// TIA Portal project "AutoCrib_StMartin" (V19)

(* hardware
DEVICE "S7-1200 station_1"  S7-1200 Station
   slot 0: "Rack_0"  S7-1200 Rack  Rack  V1.0
   slot 1: "AutoCrib_PLC"  CPU 1215C AC/DC/Rly  6ES7 215-1BG40-0XB0  V4.6
*)

// ===== PLC "AutoCrib_PLC"  CPU 1215C AC/DC/Rly =====

VAR_GLOBAL   // PLC tag table "Tt_AdminPanel"
   "xAutomaticMode" AT %I0.5 : Bool;
   "xModeChangeButton" AT %I0.4 : Bool;
END_VAR

VAR_GLOBAL   // PLC tag table "Tt_UserPanel"
   "IX_CoinSensor" AT %I0.1 : Bool;
   "IX_Billsensor" AT %I0.3 : Bool;
   "IX_MotionSensor" AT %I0.0 : Bool;
   "IX_CoinSensorCrib" AT %I0.2 : Bool;
END_VAR

VAR_GLOBAL   // PLC tag table "Tt_LightGroups"
   "QX_MinimalLightGroup" AT %Q0.0 : Bool;
   "QX_MinimalPlusLightGroup" AT %Q0.1 : Bool;
   "QX_LightGroup1" AT %Q0.2 : Bool;
   "QX_LightGroup2" AT %Q0.3 : Bool;
   "QX_LightGroup3" AT %Q0.4 : Bool;
   "QX_LightGroup4" AT %Q0.5 : Bool;
   "QX_LightGroup5" AT %Q0.6 : Bool;
   "QX_LightGroup6" AT %Q0.7 : Bool;
   "QX_LightGroup7" AT %Q1.0 : Bool;
   "QX_LightGroup_Fire" AT %Q1.1 : Bool;
END_VAR

TYPE "DT_TimeConfig"
   STRUCT
      TOD_WakeUpTime : Time_Of_Day := TOD#08:00:00;
      TOD_SleepTime : Time_Of_Day := TOD#20:00:00;
   END_STRUCT;
END_TYPE

DATA_BLOCK "DB_Global_Time"   // DB2
{ S7_Optimized_Access := 'TRUE' }
VERSION : 0.1
   VAR
      DTL_CurrentTime : DTL;
      currentDate : Date;
      TOD_CurrentTime : Time_Of_Day;
      iDayTimeError : Int;
      xDayTime : Bool := False;
      tCycleTimePT : Time := T#20S;
      tShortCycleTimePT : Time := T#2S;
      tNoMotionTimeOut : Time := T#100S;
      tSystemEnable : "DT_TimeConfig";
   END_VAR
BEGIN
   tSystemEnable.TOD_WakeUpTime := TOD#08:00:00;
   tSystemEnable.TOD_SleepTime := TOD#19:00:00;
END_DATA_BLOCK

DATA_BLOCK "DB_Global_Config"   // DB8
{ S7_Optimized_Access := 'TRUE' }
VERSION : 0.1
BEGIN
END_DATA_BLOCK

// folder: FunctionBlocks

DATA_BLOCK "FB_Time_Update_DB"   // DB1
{ S7_Optimized_Access := 'TRUE' }
VERSION : 0.1
// stored: InstanceOfName FB_Time_Update
"FB_Time_Update"
BEGIN
END_DATA_BLOCK

// folder: FunctionBlocks/MainStateMachine

DATA_BLOCK "FB_MainStateMachine_DB"   // DB7
{ S7_Optimized_Access := 'TRUE' }
VERSION : 0.1
// stored: InstanceOfName FB_MainStateMachine
"FB_MainStateMachine"
BEGIN
END_DATA_BLOCK

// folder: System blocks/Program resources

DATA_BLOCK "IEC_Timer_0_DB_AutoChangeLighting"   // DB6
{ S7_Optimized_Access := 'TRUE' }
AUTHOR : Simatic
FAMILY : IEC
NAME : IEC_TMR
VERSION : 1.0
// stored: InstanceOfName IEC_TIMER
"IEC_TIMER"
BEGIN
END_DATA_BLOCK

// folder: (top level)

FUNCTION "checkForChristmas" : Bool   // FC1, SCL
{ S7_Optimized_Access := 'TRUE' }
VERSION : 0.1
   VAR_INPUT
      inputDate : Date;
   END_VAR
   VAR_TEMP
      iCurrentDate : Int;
      iCurrentMonth : Int;
      iCurrentDay : Int;
   END_VAR
BEGIN
   #iCurrentDate := DATE_TO_INT(#inputDate);

   // Extract month and day
   #iCurrentMonth := (#iCurrentDate / 100) MOD 100;  // Get the month (MM)
   #iCurrentDay := #iCurrentDate MOD 100;  // Get the day (DD)

   // Check if the date is December 24th
   IF (#iCurrentMonth = 12) AND (#iCurrentDay = 24) THEN
       // Date is December 24th
       #checkForChristmas := TRUE;
   END_IF;
END_FUNCTION

ORGANIZATION_BLOCK "Main"   // OB1, LAD, ProgramCycle
TITLE = "Main Program Sweep (Cycle)"
{ S7_Optimized_Access := 'TRUE' }
VERSION : 0.1
// Copyright to - B.Eng Ben Cloos - ben(at)cloosefamill.lu
   VAR_INPUT
      Initial_Call : Bool;   // Initial call of this OB
      Remanence : Bool;   // =True, if remanent data are available
   END_VAR
   VAR_TEMP
      xRT_CoinSensorTriggerQ : Bool;
      xRT_BillSensorTriggerQ : Bool;
      xRT_ModeChangeTriggerQ : Bool;
      xRT_MotionTriggerQ : Bool;
      b_IsChristmas : Bool;
   END_VAR
BEGIN

REGION Network 1: Update Time every Cycle
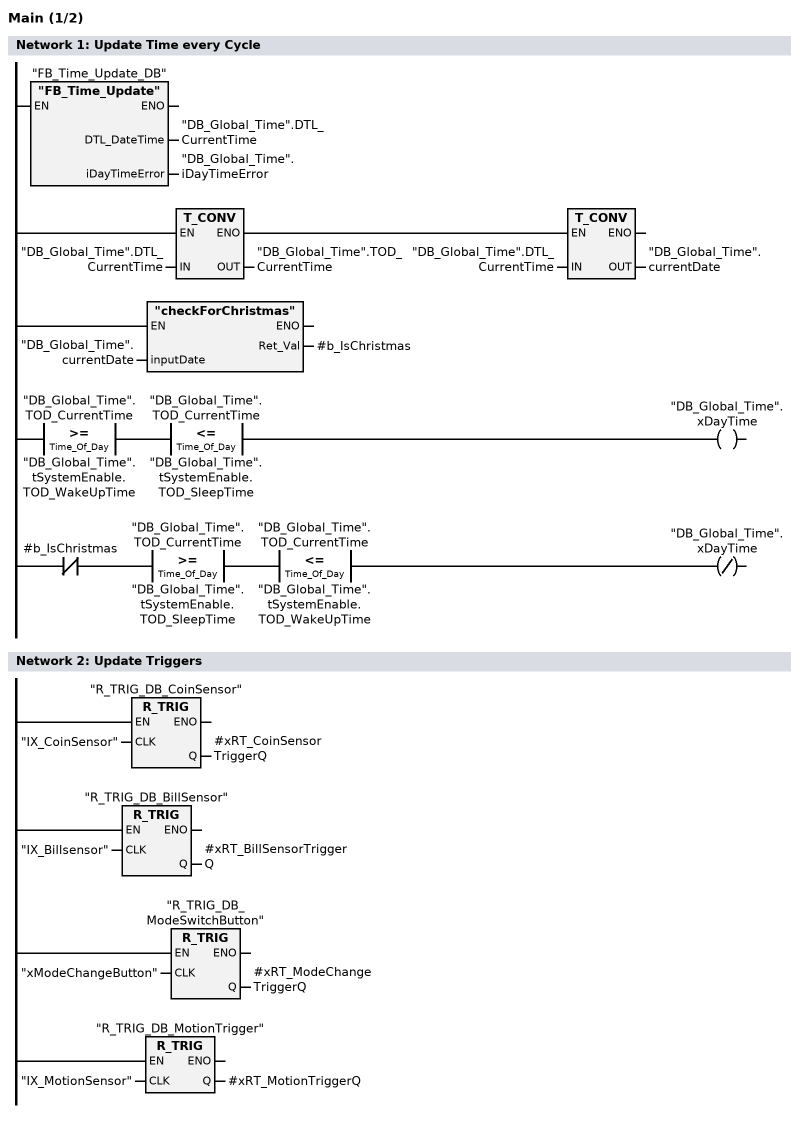
   // ENO of a box is taken as its EN; it also drops when the box reports an error
   "FB_Time_Update_DB"(DTL_DateTime => "DB_Global_Time".DTL_CurrentTime,   // "FB_Time_Update"
                       iDayTimeError => "DB_Global_Time".iDayTimeError);
   "DB_Global_Time".TOD_CurrentTime := T_CONV(IN := "DB_Global_Time".DTL_CurrentTime);
   "DB_Global_Time".currentDate := T_CONV(IN := "DB_Global_Time".DTL_CurrentTime);
   #b_IsChristmas := "checkForChristmas"(inputDate := "DB_Global_Time".currentDate);
   "DB_Global_Time".xDayTime := ("DB_Global_Time".TOD_CurrentTime >= "DB_Global_Time".tSystemEnable.TOD_WakeUpTime) AND ("DB_Global_Time".TOD_CurrentTime <= "DB_Global_Time".tSystemEnable.TOD_SleepTime);
   "DB_Global_Time".xDayTime := NOT (NOT #b_IsChristmas AND ("DB_Global_Time".TOD_CurrentTime >= "DB_Global_Time".tSystemEnable.TOD_SleepTime) AND ("DB_Global_Time".TOD_CurrentTime <= "DB_Global_Time".tSystemEnable.TOD_WakeUpTime));
END_REGION

REGION Network 2: Update Triggers
   "R_TRIG_DB_CoinSensor"(CLK := "IX_CoinSensor", Q => #xRT_CoinSensorTriggerQ);   // R_TRIG
   "R_TRIG_DB_BillSensor"(CLK := "IX_Billsensor", Q => #xRT_BillSensorTriggerQ);   // R_TRIG
   "R_TRIG_DB_ModeSwitchButton"(CLK := "xModeChangeButton", Q => #xRT_ModeChangeTriggerQ);   // R_TRIG
   "R_TRIG_DB_MotionTrigger"(CLK := "IX_MotionSensor", Q => #xRT_MotionTriggerQ);   // R_TRIG
END_REGION

REGION Network 3: State Machine Excecution
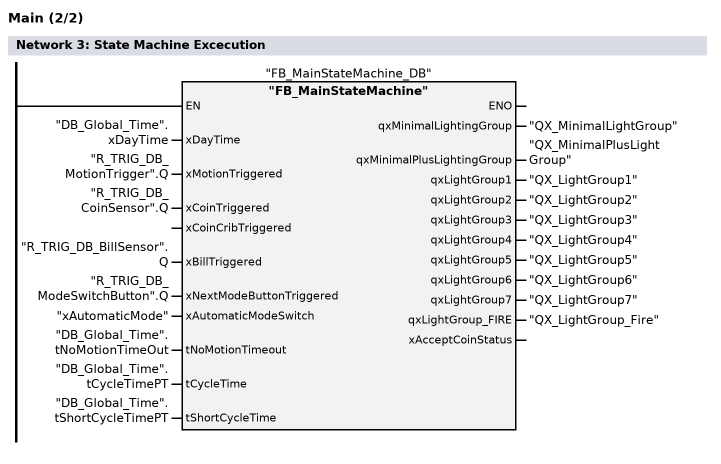
   RUNG wire#powerrail
      "FB_MainStateMachine_DB"(xDayTime := "DB_Global_Time".xDayTime, xMotionTriggered := "R_TRIG_DB_MotionTrigger".Q, xCoinTriggered := "R_TRIG_DB_CoinSensor".Q, xCoinCribTriggered :=, xBillTriggered := "R_TRIG_DB_BillSensor".Q, xNextModeButtonTriggered := "R_TRIG_DB_ModeSwitchButton".Q, xAutomaticModeSwitch := "xAutomaticMode", tNoMotionTimeout := "DB_Global_Time".tNoMotionTimeOut, tCycleTime := "DB_Global_Time".tCycleTimePT, tShortCycleTime := "DB_Global_Time".tShortCycleTimePT, qxMinimalLightingGroup => "QX_MinimalLightGroup", qxMinimalPlusLightingGroup => "QX_MinimalPlusLightGroup", qxLightGroup1 => "QX_LightGroup1", qxLightGroup2 => "QX_LightGroup2", qxLightGroup3 => "QX_LightGroup3", qxLightGroup4 => "QX_LightGroup4", qxLightGroup5 => "QX_LightGroup5", qxLightGroup6 => "QX_LightGroup6", qxLightGroup7 => "QX_LightGroup7", qxLightGroup_FIRE => "QX_LightGroup_Fire", xAcceptCoinStatus =>)
   END_RUNG
   // the same network as SCL:
   "FB_MainStateMachine_DB"(xDayTime := "DB_Global_Time".xDayTime,   // "FB_MainStateMachine"
                           xMotionTriggered := "R_TRIG_DB_MotionTrigger".Q,
                           xCoinTriggered := "R_TRIG_DB_CoinSensor".Q,
                           xBillTriggered := "R_TRIG_DB_BillSensor".Q,
                           xNextModeButtonTriggered := "R_TRIG_DB_ModeSwitchButton".Q,
                           xAutomaticModeSwitch := "xAutomaticMode",
                           tNoMotionTimeout := "DB_Global_Time".tNoMotionTimeOut,
                           tCycleTime := "DB_Global_Time".tCycleTimePT,
                           tShortCycleTime := "DB_Global_Time".tShortCycleTimePT,
                           qxMinimalLightingGroup => "QX_MinimalLightGroup",
                           qxMinimalPlusLightingGroup => "QX_MinimalPlusLightGroup",
                           qxLightGroup1 => "QX_LightGroup1",
                           qxLightGroup2 => "QX_LightGroup2",
                           qxLightGroup3 => "QX_LightGroup3",
                           qxLightGroup4 => "QX_LightGroup4",
                           qxLightGroup5 => "QX_LightGroup5",
                           qxLightGroup6 => "QX_LightGroup6",
                           qxLightGroup7 => "QX_LightGroup7",
                           qxLightGroup_FIRE => "QX_LightGroup_Fire");
END_REGION
END_ORGANIZATION_BLOCK

// folder: FunctionBlocks

FUNCTION_BLOCK "FB_Time_Update"   // FB1, SCL
{ S7_Optimized_Access := 'TRUE' }
VERSION : 0.1
   VAR_OUTPUT
      DTL_DateTime : DTL;
      iDayTimeError : Int;
   END_VAR
BEGIN
   #iDayTimeError := RD_LOC_T(OUT => #DTL_DateTime);
END_FUNCTION_BLOCK

// folder: FunctionBlocks/MainStateMachine

FUNCTION_BLOCK "FB_MainStateMachine"   // FB2, SCL
{ S7_Optimized_Access := 'TRUE' }
VERSION : 0.1
   VAR_INPUT
      xDayTime : Bool;
      xMotionTriggered : Bool;
      xCoinTriggered : Bool;
      xCoinCribTriggered : Bool;
      xBillTriggered : Bool;
      xNextModeButtonTriggered : Bool;
      xAutomaticModeSwitch : Bool;
      tNoMotionTimeout : Time;
      tCycleTime : Time;
      tShortCycleTime : Time;
   END_VAR
   VAR_OUTPUT
      qxMinimalLightingGroup : Bool;
      qxMinimalPlusLightingGroup : Bool;
      qxLightGroup1 : Bool;
      qxLightGroup2 : Bool;
      qxLightGroup3 : Bool;
      qxLightGroup4 : Bool;
      qxLightGroup5 : Bool;   // not defined
      qxLightGroup6 : Bool;   // not defined
      qxLightGroup7 : Bool;   // not defined
      qxLightGroup_FIRE : Bool;
      xAcceptCoinStatus : Bool := true;
   END_VAR
   VAR
      usi_CurrentState : USInt;
      xEntry : Bool := true;
      tCycleTimer : TON_TIME;
      tShortCycleTimer : TON_TIME;
      tNoMotionTimer : TON_TIME;
      xEnableCycleTimer : Bool := false;
      xEnableShortCycleTimer : Bool := false;
      xEnableNoMotionTimer : Bool := false;
      RT_AutomatocModeTrigger : R_TRIG;
   END_VAR
   VAR_TEMP
      xNextState_Demo : Bool;   // button and not automatic mode
   END_VAR
   VAR CONSTANT
      INIT : USInt;
      OFF : USInt := 1;
      FULL : USInt := 2;
      MINIMUM : USInt := 3;
      MINIMUM_MOTION : USInt := 4;
      LIGHTCYCLE_1 : USInt := 5;
      LIGHTCYCLE_2 : USInt := 6;
      LIGHTCYCLE_3 : USInt := 7;
      LIGHTCYCLE_4 : USInt := 8;
      LIGHTCYCLE_5 : USInt := 9;
      LIGHTCYCLE_6 : USInt := 10;
      LIGHTCYCLE_7 : USInt := 11;
      LIGHTCYCLE_8 : USInt := 12;
      LIGHTCYCLE_9 : USInt := 13;
      LIGHTCYCLE_10 : USInt := 14;
      LIGHTCYCLE_11 : USInt := 15;
      LIGHTCYCLE_12 : USInt := 16;
   END_VAR
BEGIN
   // Copyright (c) [2024] Ben Cloos, B.Eng.
   // 
   // Permission to use, copy, modify, and distribute this software for any
   // purpose with or without fee is hereby granted, provided that the above 
   // copyright notice and this permission notice appear in all copies.
   // 
   // THE SOFTWARE IS PROVIDED "AS IS" WITHOUT WARRANTY OF ANY KIND.
   // 
   // Author: Ben Cloos
   // Contact: ben@cloosefamill.lu


   //Timer calls
   #tCycleTimer(IN := #xEnableCycleTimer,
                PT := #tCycleTime);
   #tShortCycleTimer(IN := #xEnableShortCycleTimer,
                     PT := #tShortCycleTime);
   #tNoMotionTimer(IN := #xEnableNoMotionTimer,
                       PT := #tNoMotionTimeout);

   //- - - - - - - - - - - - - - - - - - - - - - - - - - - - - - - - - - - - - - - - - - - - - - - - 

   //Boolsche Variablenzusammenhänge
   #xNextState_Demo := #xNextModeButtonTriggered AND NOT #xAutomaticModeSwitch;


   //exiting manual mode should start in minimum motion or off
   #RT_AutomatocModeTrigger(CLK := #xAutomaticModeSwitch);
   IF #RT_AutomatocModeTrigger.Q THEN
       IF #xDayTime THEN
           #usi_CurrentState := #MINIMUM_MOTION;
       ELSIF NOT #xDayTime THEN
           #usi_CurrentState := #OFF;
       END_IF;

       #xEntry := TRUE;
   END_IF;



   //- - - - - - - - - - - - - - - - - - - - - - - - - - - - - - - - - - - - - - - - - - - - - - - - 

       // Main StateMachine!
       CASE #usi_CurrentState OF
           #INIT:
               #usi_CurrentState := #OFF;
               #xEntry := TRUE;

           //- - - - - - - - - - - - - - - - - - - - - - - - - - - - - - - - - - - - - - - - - - - - - - - - 

           #OFF:
               //ENTRY
               IF #xEntry THEN
                   #xEntry := FALSE;

                   #qxMinimalLightingGroup := FALSE;
                   #qxMinimalPlusLightingGroup := FALSE;
                   #qxLightGroup_FIRE := FALSE;

                   #qxLightGroup1 := FALSE;
                   #qxLightGroup2 := FALSE;
                   #qxLightGroup3 := FALSE;
                   #qxLightGroup4 := FALSE;
                   #qxLightGroup5 := FALSE;
                   #qxLightGroup6 := FALSE;
                   #qxLightGroup7 := FALSE;

               END_IF;

               //DO


               //EXIT
               //Exit Condition 1
               IF #xNextState_Demo THEN
                   #usi_CurrentState := #FULL;
                   #xEntry := TRUE;
               END_IF;
               //Exit Condition 2
               IF #xDayTime AND #xAutomaticModeSwitch THEN
                   #usi_CurrentState := #MINIMUM_MOTION;
                   #xEntry := TRUE;
               END_IF;

               //- - - - - - - - - - - - - - - - - - - - - - - - - - - - - - - - - - - - - - - - - - - - - - - - 

           #FULL:
               //entry
               IF #xEntry THEN
                   #xEntry := FALSE;

                   #qxMinimalLightingGroup := TRUE;
                   #qxMinimalPlusLightingGroup := TRUE;
                   #qxLightGroup_FIRE := TRUE;

                   #qxLightGroup1 := TRUE;
                   #qxLightGroup2 := TRUE;
                   #qxLightGroup3 := TRUE;
                   #qxLightGroup4 := TRUE;
                   #qxLightGroup5 := TRUE;
                   #qxLightGroup6 := TRUE;
                   #qxLightGroup7 := TRUE;

               END_IF;

               //DO
               //

               //EXIT
               IF #xNextState_Demo THEN
                   #xEntry := TRUE;
                   #usi_CurrentState := #MINIMUM;
               END_IF;

               //- - - - - - - - - - - - - - - - - - - - - - - - - - - - - - - - - - - - - - - - - - - - - - - - 

           #MINIMUM:
               //ENTRY
               IF #xEntry THEN
                   #xEntry := FALSE;

                   //Set Minimum Lighting!
                   #qxMinimalLightingGroup := TRUE;
                   #qxMinimalPlusLightingGroup := FALSE;
                   #qxLightGroup_FIRE := FALSE;

                   #qxLightGroup1 := FALSE;
                   #qxLightGroup2 := FALSE;
                   #qxLightGroup3 := FALSE;
                   #qxLightGroup4 := FALSE;
                   #qxLightGroup5 := FALSE;
                   #qxLightGroup6 := FALSE;
                   #qxLightGroup7 := FALSE;
               END_IF;

               //DO


               //EXIT
               //Exit Confition 1
               IF NOT #xDayTime AND #xAutomaticModeSwitch THEN
                   #xEntry := TRUE;
                   #usi_CurrentState := #OFF;
               END_IF;
               //Exit Condition 2
               IF #xNextState_Demo OR (#xDayTime AND #xMotionTriggered AND #xAutomaticModeSwitch) THEN
                   #xEntry := TRUE;
                   #usi_CurrentState := #MINIMUM_MOTION;
               END_IF;

               //- - - - - - - - - - - - - - - - - - - - - - - - - - - - - - - - - - - - - - - - - - - - - - - - 


           #MINIMUM_MOTION:
               //Entry
               IF #xEntry THEN
                   #xEntry := FALSE;
                   #xAcceptCoinStatus := TRUE; //Feedback light for user

                   //Start Motion Timer
                   #xEnableNoMotionTimer := TRUE;

                   //Set Motion Lighing!
                   #qxMinimalLightingGroup := TRUE;
                   #qxMinimalPlusLightingGroup := TRUE;
                   #qxLightGroup_FIRE := TRUE;

                   #qxLightGroup1 := FALSE;
                   #qxLightGroup2 := FALSE;
                   #qxLightGroup3 := FALSE;
                   #qxLightGroup4 := FALSE;
                   #qxLightGroup5 := FALSE;
                   #qxLightGroup6 := FALSE;
                   #qxLightGroup7 := FALSE;
               END_IF;

               //DO
               //Restart MotionTimer on motion
               IF #xMotionTriggered THEN
                   #tNoMotionTimer(IN := FALSE,
                                   PT := #tNoMotionTimeout); // called to really reset the timer!
                   #xEnableNoMotionTimer := TRUE; //not changed, written for understanding purposes
               END_IF;


               //EXIT
               //Exit Condition 1 - no motion
               IF NOT #xMotionTriggered AND #tNoMotionTimer.Q AND #xAutomaticModeSwitch THEN
                   #xEntry := TRUE;
                   #usi_CurrentState := #MINIMUM;
                   #xEnableNoMotionTimer := FALSE;
                   #xAcceptCoinStatus := FALSE;
               END_IF;
               //Exit Condition 2 - coin in lightning
               IF #xNextState_Demo OR (#xAutomaticModeSwitch AND (#xBillTriggered OR #xCoinTriggered)) THEN
                   #xEntry := TRUE;
                   #usi_CurrentState := #LIGHTCYCLE_1;
                   #xEnableNoMotionTimer := FALSE;
                   #xAcceptCoinStatus := FALSE;
               END_IF;

               //- - - - - - - - - - - - - - - - - - - - - - - - - - - - - - - - - - - - - - - - - - - - - - - - 


           #LIGHTCYCLE_1:
               IF #xEntry THEN
                   #xEntry := FALSE;
                   //Set Lighting
                   #qxMinimalLightingGroup := FALSE;
                   #qxMinimalPlusLightingGroup := FALSE;
                   #qxLightGroup_FIRE := TRUE;

                   #qxLightGroup1 := TRUE;
                   #qxLightGroup2 := FALSE;
                   #qxLightGroup3 := FALSE;
                   #qxLightGroup4 := FALSE;
                   #qxLightGroup5 := FALSE;
                   #qxLightGroup6 := FALSE;
                   #qxLightGroup7 := FALSE;

                   //Start Timer
                   IF #xAutomaticModeSwitch THEN
                       #xEnableCycleTimer := TRUE;
                   END_IF;
               END_IF;

               //DO


               //EXIT
               IF (#tCycleTimer.Q AND #xAutomaticModeSwitch) OR #xNextState_Demo THEN
                   #xEntry := TRUE;
                   #xEnableCycleTimer := FALSE;
                   #usi_CurrentState := #LIGHTCYCLE_2;
               END_IF;

               //- - - - - - - - - - - - - - - - - - - - - - - - - - - - - - - - - - - - - - - - - - - - - - - - 


           #LIGHTCYCLE_2:
               IF #xEntry THEN
                   #xEntry := FALSE;
                   //Set Lighting
                   #qxMinimalLightingGroup := FALSE;
                   #qxMinimalPlusLightingGroup := FALSE;
                   #qxLightGroup_FIRE := TRUE;

                   #qxLightGroup1 := FALSE;
                   #qxLightGroup2 := TRUE;
                   #qxLightGroup3 := FALSE;
                   #qxLightGroup4 := FALSE;
                   #qxLightGroup5 := FALSE;
                   #qxLightGroup6 := FALSE;
                   #qxLightGroup7 := FALSE;

                   //Start Timer
                   IF #xAutomaticModeSwitch THEN
                       #xEnableCycleTimer := TRUE;
                   END_IF;
               END_IF;

               //DO


               //EXIT
               IF (#tCycleTimer.Q AND #xAutomaticModeSwitch) OR #xNextState_Demo THEN
                   #xEntry := TRUE;
                   #xEnableCycleTimer := FALSE;
                   #usi_CurrentState := #LIGHTCYCLE_3;
               END_IF;

               //- - - - - - - - - - - - - - - - - - - - - - - - - - - - - - - - - - - - - - - - - - - - - - - - 


           #LIGHTCYCLE_3:
               IF #xEntry THEN
                   #xEntry := FALSE;
                   //Set Lighting
                   #qxMinimalLightingGroup := FALSE;
                   #qxMinimalPlusLightingGroup := FALSE;
                   #qxLightGroup_FIRE := TRUE;

                   #qxLightGroup1 := FALSE;
                   #qxLightGroup2 := FALSE;
                   #qxLightGroup3 := TRUE;
                   #qxLightGroup4 := FALSE;
                   #qxLightGroup5 := FALSE;
                   #qxLightGroup6 := FALSE;
                   #qxLightGroup7 := FALSE;

                   //Start Timer
                   IF #xAutomaticModeSwitch THEN
                       #xEnableCycleTimer := TRUE;
                   END_IF;
               END_IF;

               //DO


               //EXIT
               IF (#tCycleTimer.Q AND #xAutomaticModeSwitch) OR #xNextState_Demo THEN
                   #xEntry := TRUE;
                   #xEnableCycleTimer := FALSE;
                   #usi_CurrentState := #LIGHTCYCLE_4;
               END_IF;

               //- - - - - - - - - - - - - - - - - - - - - - - - - - - - - - - - - - - - - - - - - - - - - - - - 


           #LIGHTCYCLE_4:
               IF #xEntry THEN
                   #xEntry := FALSE;
                   //Set Lighting
                   #qxMinimalLightingGroup := FALSE;
                   #qxMinimalPlusLightingGroup := FALSE;
                   #qxLightGroup_FIRE := TRUE;

                   #qxLightGroup1 := FALSE;
                   #qxLightGroup2 := FALSE;
                   #qxLightGroup3 := FALSE;
                   #qxLightGroup4 := TRUE;
                   #qxLightGroup5 := FALSE;
                   #qxLightGroup6 := FALSE;
                   #qxLightGroup7 := FALSE;

                   //Start Timer
                   IF #xAutomaticModeSwitch THEN
                       #xEnableCycleTimer := TRUE;
                   END_IF;
               END_IF;

               //DO


               //EXIT
               IF (#tCycleTimer.Q AND #xAutomaticModeSwitch) OR #xNextState_Demo THEN
                   #xEntry := TRUE;
                   #xEnableCycleTimer := FALSE;
                   #usi_CurrentState := #LIGHTCYCLE_5;
               END_IF;

               //- - - - - - - - - - - - - - - - - - - - - - - - - - - - - - - - - - - - - - - - - - - - - - - - 


           #LIGHTCYCLE_5:
               IF #xEntry THEN
                   #xEntry := FALSE;
                   //Set Lighting
                   #qxMinimalLightingGroup := FALSE;
                   #qxMinimalPlusLightingGroup := FALSE;
                   #qxLightGroup_FIRE := TRUE;

                   #qxLightGroup1 := FALSE;
                   #qxLightGroup2 := FALSE;
                   #qxLightGroup3 := TRUE;
                   #qxLightGroup4 := TRUE;
                   #qxLightGroup5 := FALSE;
                   #qxLightGroup6 := FALSE;
                   #qxLightGroup7 := FALSE;

                   //Start Timer
                   IF #xAutomaticModeSwitch THEN
                       #xEnableCycleTimer := TRUE;
                   END_IF;
               END_IF;

               //DO


               //EXIT
               IF (#tCycleTimer.Q AND #xAutomaticModeSwitch) OR #xNextState_Demo THEN
                   #xEntry := TRUE;
                   #xEnableCycleTimer := FALSE;
                   #usi_CurrentState := #LIGHTCYCLE_6;
               END_IF;

               //- - - - - - - - - - - - - - - - - - - - - - - - - - - - - - - - - - - - - - - - - - - - - - - - 


           #LIGHTCYCLE_6:
               IF #xEntry THEN
                   #xEntry := FALSE;
                   //Set Lighting
                   #qxMinimalLightingGroup := FALSE;
                   #qxMinimalPlusLightingGroup := FALSE;
                   #qxLightGroup_FIRE := TRUE;

                   #qxLightGroup1 := FALSE;
                   #qxLightGroup2 := TRUE;
                   #qxLightGroup3 := TRUE;
                   #qxLightGroup4 := TRUE;
                   #qxLightGroup5 := FALSE;
                   #qxLightGroup6 := FALSE;
                   #qxLightGroup7 := FALSE;

                   //Start Timer
                   IF #xAutomaticModeSwitch THEN
                       #xEnableCycleTimer := TRUE;
                   END_IF;
               END_IF;

               //DO


               //EXIT
               IF (#tCycleTimer.Q AND #xAutomaticModeSwitch) OR #xNextState_Demo THEN
                   #xEntry := TRUE;
                   #xEnableCycleTimer := FALSE;
                   #usi_CurrentState := #LIGHTCYCLE_7;
               END_IF;

               //- - - - - - - - - - - - - - - - - - - - - - - - - - - - - - - - - - - - - - - - - - - - - - - - 


           #LIGHTCYCLE_7:
               IF #xEntry THEN
                   #xEntry := FALSE;
                   //Set Lighting
                   #qxMinimalLightingGroup := FALSE;
                   #qxMinimalPlusLightingGroup := FALSE;
                   #qxLightGroup_FIRE := TRUE;

                   #qxLightGroup1 := TRUE;
                   #qxLightGroup2 := TRUE;
                   #qxLightGroup3 := TRUE;
                   #qxLightGroup4 := TRUE;
                   #qxLightGroup5 := FALSE;
                   #qxLightGroup6 := FALSE;
                   #qxLightGroup7 := FALSE;

                   //Start Timer
                   IF #xAutomaticModeSwitch THEN
                       #xEnableCycleTimer := TRUE;
                   END_IF;
               END_IF;

               //DO


               //EXIT
               IF (#tCycleTimer.Q AND #xAutomaticModeSwitch) OR #xNextState_Demo THEN
                   #xEntry := TRUE;
                   #xEnableCycleTimer := FALSE;
                   #usi_CurrentState := #LIGHTCYCLE_8;
               END_IF;

               //- - - - - - - - - - - - - - - - - - - - - - - - - - - - - - - - - - - - - - - - - - - - - - - - 


           #LIGHTCYCLE_8:
               IF #xEntry THEN
                   #xEntry := FALSE;
                   //Set Lighting
                   #qxMinimalLightingGroup := TRUE;
                   #qxMinimalPlusLightingGroup := TRUE;
                   #qxLightGroup_FIRE := TRUE;

                   #qxLightGroup1 := FALSE;
                   #qxLightGroup2 := TRUE;
                   #qxLightGroup3 := TRUE;
                   #qxLightGroup4 := TRUE;
                   #qxLightGroup5 := FALSE;
                   #qxLightGroup6 := FALSE;
                   #qxLightGroup7 := FALSE;

                   //Start Timer
                   IF #xAutomaticModeSwitch THEN
                       #xEnableCycleTimer := TRUE;
                   END_IF;
               END_IF;

               //DO


               //EXIT
               IF (#tCycleTimer.Q AND #xAutomaticModeSwitch) OR #xNextState_Demo THEN
                   #xEntry := TRUE;
                   #xEnableCycleTimer := FALSE;
                   #usi_CurrentState := #LIGHTCYCLE_9;
               END_IF;

               //- - - - - - - - - - - - - - - - - - - - - - - - - - - - - - - - - - - - - - - - - - - - - - - - 


           #LIGHTCYCLE_9:
               IF #xEntry THEN
                   #xEntry := FALSE;
                   //Set Lighting
                   #qxMinimalLightingGroup := TRUE;
                   #qxMinimalPlusLightingGroup := TRUE;
                   #qxLightGroup_FIRE := TRUE;

                   #qxLightGroup1 := FALSE;
                   #qxLightGroup2 := FALSE;
                   #qxLightGroup3 := TRUE;
                   #qxLightGroup4 := TRUE;
                   #qxLightGroup5 := FALSE;
                   #qxLightGroup6 := FALSE;
                   #qxLightGroup7 := FALSE;

                   //Start Timer
                   IF #xAutomaticModeSwitch THEN
                       #xEnableShortCycleTimer := TRUE;
                   END_IF;
               END_IF;

               //DO


               //EXIT
               IF (#tShortCycleTimer.Q AND #xAutomaticModeSwitch) OR #xNextState_Demo THEN
                   #xEntry := TRUE;
                   #xEnableShortCycleTimer := FALSE;
                   #usi_CurrentState := #LIGHTCYCLE_10;
               END_IF;

               //- - - - - - - - - - - - - - - - - - - - - - - - - - - - - - - - - - - - - - - - - - - - - - - - 


           #LIGHTCYCLE_10:
               IF #xEntry THEN
                   #xEntry := FALSE;
                   //Set Lighting
                   #qxMinimalLightingGroup := TRUE;
                   #qxMinimalPlusLightingGroup := TRUE;
                   #qxLightGroup_FIRE := TRUE;

                   #qxLightGroup1 := FALSE;
                   #qxLightGroup2 := FALSE;
                   #qxLightGroup3 := FALSE;
                   #qxLightGroup4 := TRUE;
                   #qxLightGroup5 := FALSE;
                   #qxLightGroup6 := FALSE;
                   #qxLightGroup7 := FALSE;

                   //Start Timer
                   IF #xAutomaticModeSwitch THEN
                       #xEnableShortCycleTimer := TRUE;
                   END_IF;
               END_IF;

               //DO


               //EXIT
               IF (#tShortCycleTimer.Q AND #xAutomaticModeSwitch) OR #xNextState_Demo THEN
                   #xEntry := TRUE;
                   #xEnableShortCycleTimer := FALSE;
                   #usi_CurrentState := #LIGHTCYCLE_11;
               END_IF;

               //- - - - - - - - - - - - - - - - - - - - - - - - - - - - - - - - - - - - - - - - - - - - - - - - 


           #LIGHTCYCLE_11:
               IF #xEntry THEN
                   #xEntry := FALSE;
                   //Set Lighting
                   #qxMinimalLightingGroup := TRUE;
                   #qxMinimalPlusLightingGroup := TRUE;
                   #qxLightGroup_FIRE := TRUE;

                   #qxLightGroup1 := FALSE;
                   #qxLightGroup2 := FALSE;
                   #qxLightGroup3 := FALSE;
                   #qxLightGroup4 := FALSE;
                   #qxLightGroup5 := FALSE;
                   #qxLightGroup6 := FALSE;
                   #qxLightGroup7 := FALSE;

                   //Start Timer
                   IF #xAutomaticModeSwitch THEN
                       #xEnableShortCycleTimer := TRUE;
                   END_IF;
               END_IF;

               //DO


               //EXIT
               IF (#tShortCycleTimer.Q AND #xAutomaticModeSwitch) OR #xNextState_Demo THEN
                   #xEntry := TRUE;
                   #xEnableShortCycleTimer := FALSE;
                   #usi_CurrentState := #MINIMUM_MOTION;
               END_IF;

       END_CASE;
END_FUNCTION_BLOCK